// TIA Portal V19 export
DATA_BLOCK "LineStates_DB"   // DB9
// stored: InstanceOfName LineStates, InstanceOfType FB
"LineStates"
   // VAR
   //    StateM1LineRunning { S7_SetPoint := 'True'} : "GenericState";
   //    StateM2LineRunning { S7_SetPoint := 'True'} : "GenericState";
   //    StateM1CurrentOrderNo { S7_SetPoint := 'True'} : "GenericState";
   //    StateM2CurrentOrderNo { S7_SetPoint := 'True'} : "GenericState";
   //    PubJsonMqttInstM1LineRunning { S7_SetPoint := 'True'} : "PublishJsonMqtt";
   //    PubJsonMqttInstM2LineRunning { S7_SetPoint := 'True'} : "PublishJsonMqtt";
   //    PubJsonMqttInstM1CurrentOrderNo { S7_SetPoint := 'True'} : "PublishJsonMqtt";
   //    PubJsonMqttInstM2CurrentOrderNo { S7_SetPoint := 'True'} : "PublishJsonMqtt";
   //    tpGen01 { S7_SetPoint := 'True'} : TP_TIME;
   //    tpGen02 { S7_SetPoint := 'True'} : TP_TIME;
   // END_VAR
BEGIN
END_DATA_BLOCK
